{attribute 'GeneratedUsingTerminal: EK1122-0000-0018'}
{attribute addProperty BoxType "EK1122-0000-0018"}
{attribute addProperty Id "Beckhoff_EL99xxsub_EK1100EK1100_AB5A94672"}
{attribute addProperty CRC "2229475521"}
{attribute addProperty Size "2"}
TYPE Beckhoff_EL99xxEK1122_84E318C1 EXTENDS EK1122_AB5A9467 :
STRUCT
	{attribute addProperty Name "Beckhoff_EL99xxsub_EK1100"}
	{attribute addProperty PreviousPort "Beckhoff EL99xxEK1122 : D"}
	Beckhoff_EL99xxsub_EK1100 : EK1100_AB5A9467;
END_STRUCT
END_TYPE

(* stored: Version 1.2.0.0, ProductVersion 3.1.4024.9
   DUT Beckhoff_EL99xxEK1122_84E318C1: Id {a7abe7c1-518d-4fdc-8c7f-8b68cb482d82} *)
